INTERFACE I_GigeSoftTrigger_Mode EXTENDS __SYSTEM.IQueryInterface

PROPERTY GigeCamera : I_GigEVision_Mode
GET
END_GET
SET
END_SET
END_PROPERTY

METHOD Trigger : HRESULT
VAR_INPUT
	//The data type T_DCTIME64 represents the distributed clock system time (abbreviated as DC time) as a linear 64-bit integer value. 
	//The time is expressed in nanoseconds since 1/1/2000 UTC. The smallest unit is a nanosecond.
	//F_GetCurDcTickTime64()
	nDCTimeStamp	: T_DCTIME64;
END_VAR
END_METHOD

{attribute 'monitoring' := 'call'}
PROPERTY TriggerDelay_1ns : UDINT
GET
END_GET
SET
END_SET
END_PROPERTY

END_INTERFACE

(* stored: Version 1.1.0.1, ProductVersion 3.1.4024.12
   Itf I_GigeSoftTrigger_Mode: Id {9fc15e05-923a-4f26-bd96-2504bd266e8b}
   Property GigeCamera: Id {d72b9a73-615d-4bf4-8c06-f18b484dede6}
   Get Get: Id {4f2b4bc5-1090-4a68-ae49-287cbb11a8a1}
   Set Set: Id {bc4f83ee-c487-497c-8adc-d3419a65cd16}
   Method Trigger: Id {d2062b57-95fc-4baf-9fa5-b89454f4c435}
   Property TriggerDelay_1ns: Id {b51e6435-ed51-46fd-8b6f-65d4ab29eac5}
   Get Get: Id {a5398265-c909-4aff-b1fa-8c17f6abce3c}
   Set Set: Id {0a687b8f-cf76-4123-b039-693288612315} *)
